// TIA Portal V15.1 export
// export: Created 2020-06-12T07:35:53.1630859Z, ExportSetting None, DisplayName Totally Integrated Automation Portal, DisplayVersion V15.1, DisplayName TIA Portal Openness, DisplayVersion V15.1, DisplayName STEP 7 Professional, DisplayVersion V15.1, DisplayName STEP 7 Safety, DisplayVersion V15.1, DisplayName WinCC Advanced, DisplayVersion V15.1
FUNCTION "MELT_CPS_MS" : Void   // FC172, FBD
TITLE = Meltrate+Swing controllers
{ S7_Optimized_Access := 'TRUE' }
// stored: SetENOAutomatically False
   VAR_TEMP
      tBool : Bool;
      tLim2_DelayOff : Bool;
      tLoadParam : Bool;
      tMRout : Real;
      tSWout : Real;
   END_VAR
BEGIN

REGION Network 1: Meltrate controller
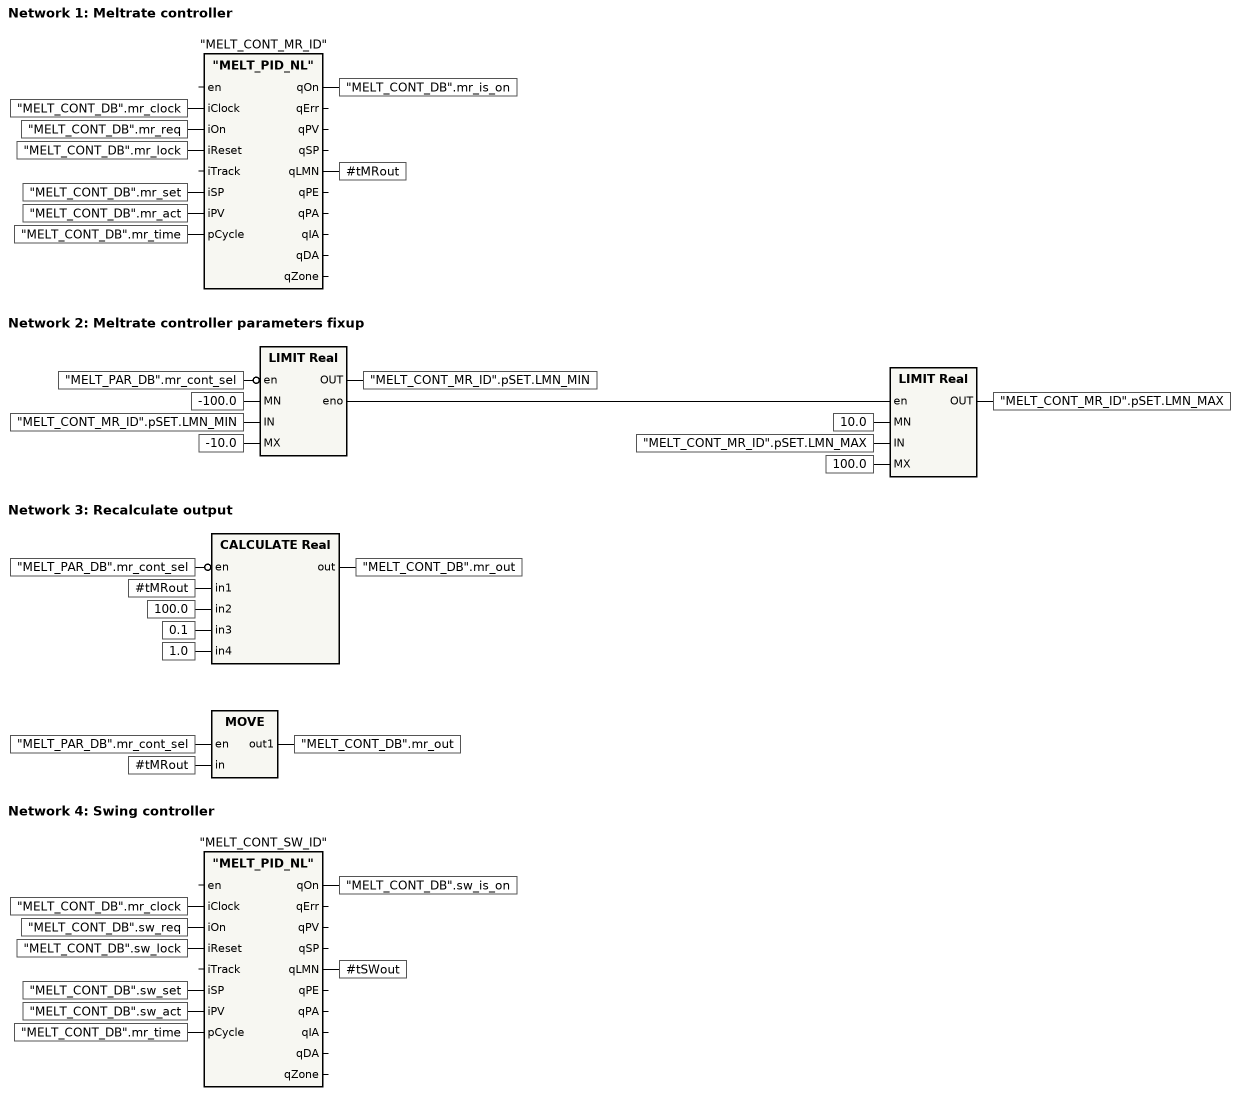
   "MELT_CONT_MR_ID"(iClock := "MELT_CONT_DB".mr_clock,   // "MELT_PID_NL"
                     iOn := "MELT_CONT_DB".mr_req,
                     iReset := "MELT_CONT_DB".mr_lock,
                     iSP := "MELT_CONT_DB".mr_set,
                     iPV := "MELT_CONT_DB".mr_act,
                     pCycle := "MELT_CONT_DB".mr_time,
                     qOn => "MELT_CONT_DB".mr_is_on,
                     qLMN => #tMRout);
END_REGION

REGION Network 2: Meltrate controller parameters fixup
   IF NOT "MELT_PAR_DB".mr_cont_sel THEN
       "MELT_CONT_MR_ID".pSET.LMN_MIN := LIMIT(MN := -100.0, IN := "MELT_CONT_MR_ID".pSET.LMN_MIN, MX := -10.0);
       "MELT_CONT_MR_ID".pSET.LMN_MAX := LIMIT(MN := 10.0, IN := "MELT_CONT_MR_ID".pSET.LMN_MAX, MX := 100.0);
   END_IF;
END_REGION

REGION Network 3: Recalculate output
   // This block allow to use 2 different calculation method:
   // 0 = Old INTECO 1.0based
   // 1 = new, with absolute value
   IF NOT "MELT_PAR_DB".mr_cont_sel THEN "MELT_CONT_DB".mr_out := 1.0+(#tMRout/100.0)*0.1; END_IF;
   IF "MELT_PAR_DB".mr_cont_sel THEN "MELT_CONT_DB".mr_out := #tMRout; END_IF;
END_REGION

REGION Network 4: Swing controller
   "MELT_CONT_SW_ID"(iClock := "MELT_CONT_DB".mr_clock,   // "MELT_PID_NL"
                     iOn := "MELT_CONT_DB".sw_req,
                     iReset := "MELT_CONT_DB".sw_lock,
                     iSP := "MELT_CONT_DB".sw_set,
                     iPV := "MELT_CONT_DB".sw_act,
                     pCycle := "MELT_CONT_DB".mr_time,
                     qOn => "MELT_CONT_DB".sw_is_on,
                     qLMN => #tSWout);
END_REGION

REGION Network 5: Swing controller parameters fixup
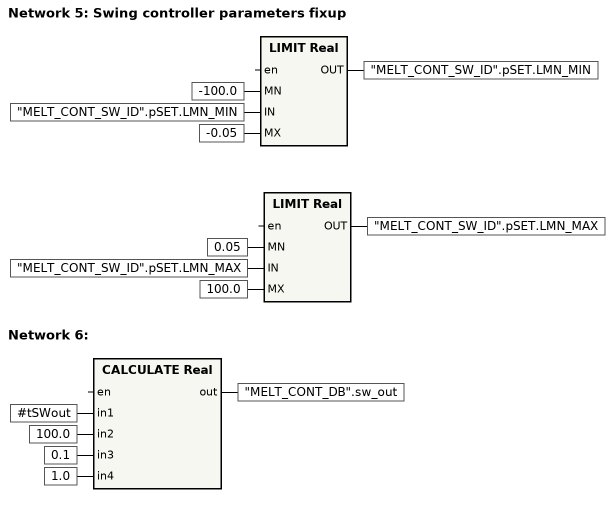
   "MELT_CONT_SW_ID".pSET.LMN_MIN := LIMIT(MN := -100.0, IN := "MELT_CONT_SW_ID".pSET.LMN_MIN, MX := -0.05);
   "MELT_CONT_SW_ID".pSET.LMN_MAX := LIMIT(MN := 0.05, IN := "MELT_CONT_SW_ID".pSET.LMN_MAX, MX := 100.0);
END_REGION

REGION Network 6
   "MELT_CONT_DB".sw_out := 1.0+(#tSWout/100.0)*0.1;
END_REGION
END_FUNCTION
